// TIA Portal project "chietrotchatlong" (V16)

(* hardware
DEVICE "S7-1200 station_1"  S7-1200 Station
   slot 0: "Rack_0"  S7-1200 Rack  Rack  V1.0
   slot 1: "PLC_1"  CPU 1214C DC/DC/DC  6ES7 214-1AG40-0XB0  V4.4
DEVICE "PC-System_1"  SIMATIC PC station
   slot 0: "SIMATIC PC station"  Rail  SIMATIC PC-Station  V1.0
      slot 125: "Stationmanager"  Station_Manager  V6.0.4
   slot 1: "HMI_RT_1"  WinCC RT Advanced  6AV2 104-0xxxx-xxxx  16.0.0.0
      slot 33792: "Computer interface"  Host interface
   slot 2: "IE general_1"  IE General  IE_CP  V8.2.0
*)

// ===== PLC "PLC_1"  CPU 1214C DC/DC/DC =====

VAR_GLOBAL   // PLC tag table "Default tag table"
   "a0" AT %M0.0 : Bool;
   "a1" AT %M0.1 : Bool;
   "b0" AT %M0.2 : Bool;
   "b1" AT %M0.3 : Bool;
   "d1" AT %M0.4 : Bool;
   "d2" AT %M0.5 : Bool;
   "d3" AT %M0.6 : Bool;
   "g" AT %M0.7 : Bool;
   "S0" AT %Q0.0 : Bool;
   "S1" AT %Q0.1 : Bool;
   "S2" AT %Q0.2 : Bool;
   "S3" AT %Q0.3 : Bool;
   "S4" AT %Q0.4 : Bool;
   "S5" AT %Q0.5 : Bool;
   "S6" AT %Q0.6 : Bool;
   "S7" AT %Q0.7 : Bool;
   "S8" AT %Q1.0 : Bool;
   "m" AT %M1.0 : Bool;
   "ThoiGian" AT %MD1 : Time;
   "START" AT %M1.1 : Bool;
   "STOP" AT %M1.2 : Bool;
   "POWER" AT %Q1.1 : Bool;
END_VAR

// folder: System blocks/Program resources

DATA_BLOCK "T2"   // DB2
{ S7_Optimized_Access := 'TRUE' }
AUTHOR : Simatic
FAMILY : IEC
NAME : IEC_TMR
VERSION : 1.0
// stored: InstanceOfName IEC_TIMER
"IEC_TIMER"
BEGIN
END_DATA_BLOCK

// folder: (top level)

ORGANIZATION_BLOCK "Main"   // OB1, FBD, ProgramCycle
TITLE = "Main Program Sweep (Cycle)"
{ S7_Optimized_Access := 'TRUE' }
VERSION : 0.1
   VAR_INPUT
      Initial_Call : Bool;   // Initial call of this OB
      Remanence : Bool;   // =True, if remanent data are available
   END_VAR
BEGIN

REGION Network 1
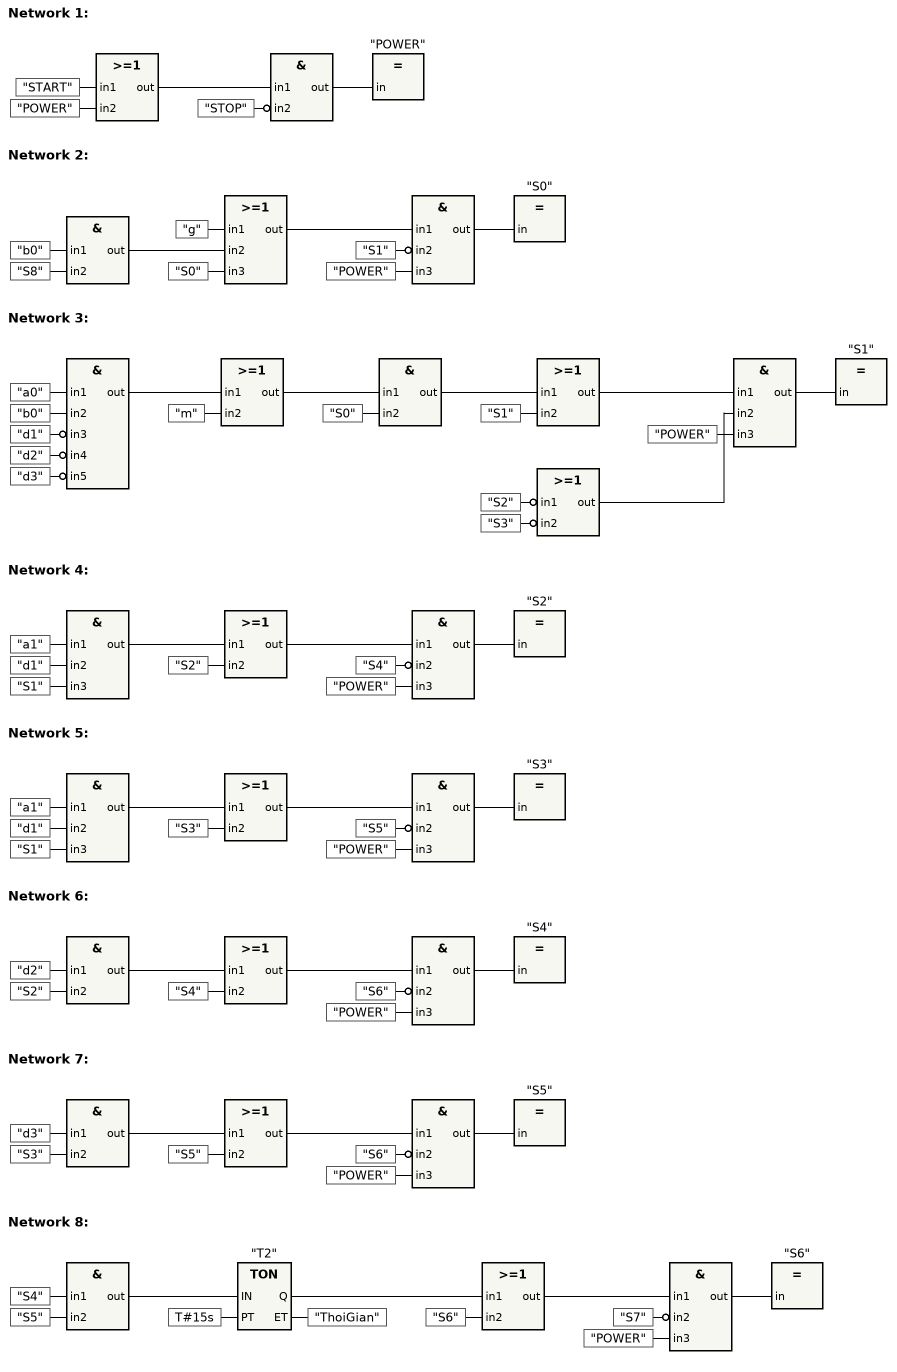
   "POWER" := ("START" OR "POWER") AND NOT "STOP";
END_REGION

REGION Network 2
   "S0" := ("g" OR ("b0" AND "S8") OR "S0") AND NOT "S1" AND "POWER";
END_REGION

REGION Network 3
   "S1" := (((("a0" AND "b0" AND NOT "d1" AND NOT "d2" AND NOT "d3") OR "m") AND "S0") OR "S1") AND (NOT "S2" OR NOT "S3") AND "POWER";
END_REGION

REGION Network 4
   "S2" := (("a1" AND "d1" AND "S1") OR "S2") AND NOT "S4" AND "POWER";
END_REGION

REGION Network 5
   "S3" := (("a1" AND "d1" AND "S1") OR "S3") AND NOT "S5" AND "POWER";
END_REGION

REGION Network 6
   "S4" := (("d2" AND "S2") OR "S4") AND NOT "S6" AND "POWER";
END_REGION

REGION Network 7
   "S5" := (("d3" AND "S3") OR "S5") AND NOT "S6" AND "POWER";
END_REGION

REGION Network 8
   "T2".TON(IN := "S4" AND "S5", PT := T#15s, ET => "ThoiGian");
   "S6" := ("T2".Q OR "S6") AND NOT "S7" AND "POWER";
END_REGION

REGION Network 9
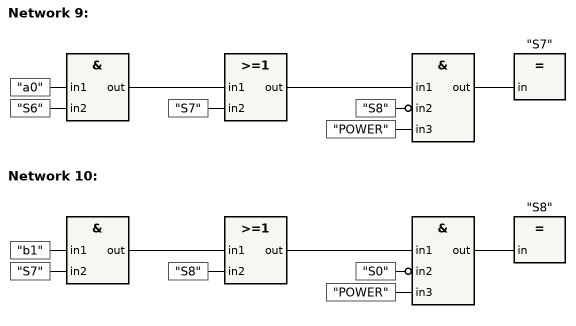
   "S7" := (("a0" AND "S6") OR "S7") AND NOT "S8" AND "POWER";
END_REGION

REGION Network 10
   "S8" := (("b1" AND "S7") OR "S8") AND NOT "S0" AND "POWER";
END_REGION
END_ORGANIZATION_BLOCK

(* ===== HMI "HMI_RT_1" =====
system functions are stored by id; their names below are inferred from use
connection "HMI_Connection_1": ETHERNET, S7_1200_OMS

HMI tags "Default tag table"
   "POWER" : Bool = PLC POWER AT %Q1.1, 1 s
   "S0" : Bool = PLC S0 AT %Q0.0, 1 s
   "S1" : Bool = PLC S1 AT %Q0.1, 1 s
   "S2" : Bool = PLC S2 AT %Q0.2, 1 s
   "S3" : Bool = PLC S3 AT %Q0.3, 1 s
   "S4" : Bool = PLC S4 AT %Q0.4, 1 s
   "S5" : Bool = PLC S5 AT %Q0.5, 1 s
   "S6" : Bool = PLC S6 AT %Q0.6, 1 s
   "S7" : Bool = PLC S7 AT %Q0.7, 1 s
   "S8" : Bool = PLC S8 AT %Q1.0, 1 s
   "START" : Bool = PLC START AT %M1.1, 1 s
   "STOP" : Bool = PLC STOP AT %M1.2, 1 s
   "a0" : Bool = PLC a0 AT %M0.0, 1 s
   "a1" : Bool = PLC a1 AT %M0.1, 1 s
   "b0" : Bool = PLC b0 AT %M0.2, 1 s
   "b1" : Bool = PLC b1 AT %M0.3, 1 s
   "d1" : Bool = PLC d1 AT %M0.4, 1 s
   "d2" : Bool = PLC d2 AT %M0.5, 1 s
   "d3" : Bool = PLC d3 AT %M0.6, 1 s
   "g" : Bool = PLC g AT %M0.7, 1 s
   "m" : Bool = PLC m AT %M1.0, 1 s
   "ThoiGian" : Time = PLC ThoiGian AT %MD1, 1 s

screen "Screen_1" 1024x768
   GraphicView "Graphic view_1" at 255,236 size 64x85; Picture "Graphic_20"
      Visibility <- "S0"
   GraphicView "Graphic view_7" at 383,148 size 56x129; Picture "Graphic_17"
      Visibility <- "S7"
   GraphicView "Graphic view_5" at 149,253 size 166x49; Picture "Graphic_14"
      Visibility <- "S1"
   Rectangle "Rectangle_1" at 721,6 size 57x26
      Appearance <- "POWER"
   Button "Button_1" at 28,15 size 64x33; TextOff 'START'
      on Press: SetBit("START")
      on Release: ResetBit("START")
   Button "Button_2" at 28,61 size 64x33; TextOff 'STOP'
      on Press: SetBit("STOP")
      on Release: ResetBit("STOP")
   Button "Button_3" at 28,107 size 64x33; TextOff 'a0'
      on Press: SetBit("a0")
      on Release: ResetBit("a0")
   Button "Button_4" at 28,153 size 64x33; TextOff 'a1'
      on Release: ResetBit("a1")
      on Press: SetBit("a1")
   Button "Button_5" at 28,199 size 64x33; TextOff 'b0'
      on Activate: SetBit("b0")
      on Deactivate: ResetBit("b0")
   Button "Button_6" at 28,245 size 64x33; TextOff 'b1'
      on Release: ResetBit("b1")
      on Press: SetBit("b1")
   Button "Button_7" at 28,291 size 64x33; TextOff 'd1'
      on Activate: SetBit("d1")
      on Deactivate: ResetBit("d1")
   Button "Button_8" at 28,337 size 64x33; TextOff 'd2'
      on Activate: SetBit("d2")
      on Deactivate: ResetBit("d2")
   Button "Button_9" at 28,383 size 64x33; TextOff 'd3'
      on Activate: SetBit("d3")
      on Deactivate: ResetBit("d3")
   Rectangle "Rectangle_2" at 721,48 size 57x26
      Appearance <- "S0"
   Rectangle "Rectangle_3" at 721,90 size 57x26
      Appearance <- "S1"
   Rectangle "Rectangle_4" at 721,132 size 57x26
      Appearance <- "S2"
   Rectangle "Rectangle_5" at 721,174 size 57x26
      Appearance <- "S3"
   Rectangle "Rectangle_6" at 721,216 size 57x26
      Appearance <- "S4"
   Rectangle "Rectangle_7" at 721,258 size 57x26
      Appearance <- "S5"
   Rectangle "Rectangle_8" at 721,300 size 57x26
      Appearance <- "S6"
   Rectangle "Rectangle_9" at 721,342 size 57x26
      Appearance <- "S7"
   Rectangle "Rectangle_10" at 721,384 size 57x26
      Appearance <- "S8"
   TextField "Text field_1" at 716,6 size 62x22; Text 'POWER'
   TextField "Text field_2" at 737,48 size 25x22; Text 'S0'
   TextField "Text field_3" at 737,91 size 25x22; Text 'S1'
   TextField "Text field_4" at 737,132 size 25x22; Text 'S2'
   TextField "Text field_5" at 737,177 size 25x22; Text 'S3'
   TextField "Text field_6" at 736,218 size 25x22; Text 'S4'
   TextField "Text field_7" at 736,262 size 25x22; Text 'S5'
   TextField "Text field_8" at 736,302 size 25x22; Text 'S6'
   TextField "Text field_9" at 736,346 size 25x22; Text 'S7'
   TextField "Text field_10" at 736,388 size 25x22; Text 'S8'
   Button "Button_10" at 28,430 size 64x33; TextOff 'g'
      on Release: ResetBit("g")
      on Press: SetBit("g")
   Button "Button_11" at 28,477 size 64x33; TextOff 'm'
      on Release: ResetBit("m")
      on Press: SetBit("m")
   GraphicView "Graphic view_4" at 127,250 size 125x50; Picture "Graphic_13"
      Visibility <- "POWER"
   GraphicView "Graphic view_16" at 386,103 size 53x120; Picture "Graphic_15"
      Visibility <- "POWER"
   Circle "Circle_1" at 611,192 size 40x40
      Appearance <- "d3"
   Circle "Circle_2" at 611,236 size 40x40
      Appearance <- "d2"
   Circle "Circle_3" at 611,278 size 40x40
      Appearance <- "d1"
   TextField "Text field_11" at 153,223 size 70x22; Text 'Xi lanh A'
   TextField "Text field_12" at 378,70 size 70x22; Text 'Xi lanh B'
   TextField "Text field_13" at 560,131 size 133x22; Text 'Các đèn cảm biến'
   GraphicView "Graphic view_2" at 376,233 size 64x85; Picture "Graphic_20"
      Visibility <- "S1"
   GraphicView "Graphic view_3" at 376,233 size 64x85; Picture "Graphic_20"
      Visibility <- "S2"
   GraphicView "Graphic view_8" at 376,233 size 64x85; Picture "Graphic_20"
      Visibility <- "S4"
   GraphicView "Graphic view_9" at 376,233 size 64x85; Picture "Graphic_20"
      Visibility <- "S5"
   TextField "Text field_14" at 452,142 size 47x22; Text 'Van C'
   TextField "Text field_15" at 315,152 size 46x22; Text 'Van E'
   GraphicView "Graphic view_12" at 287,177 size 90x59; Picture "Graphic_21"
      Appearance <- "S3"
   GraphicView "Graphic view_13" at 442,171 size 75x66; Picture "Graphic_22"
      Appearance <- "S2"
   GraphicView "Graphic view_14" at 230,202 size 60x31; Picture "Graphic_30"
   GraphicView "Graphic view_15" at 230,1 size 58x204; Picture "Graphic_31"
   GraphicView "Graphic view_17" at 512,177 size 56x75; Picture "Graphic_32"
   GraphicView "Graphic view_18" at 511,0 size 59x181; Picture "Graphic_31"
   GraphicView "Graphic view_19" at 375,346 size 64x85; Picture "Graphic_33"
      Visibility <- "S7"
   GraphicView "Graphic view_11" at 375,346 size 64x85; Picture "Graphic_33"
      Visibility <- "S8"
   GraphicView "Graphic view_20" at 376,233 size 64x85; Picture "Graphic_7"
      Visibility <- "S3"
   GraphicView "Graphic view_21" at 376,233 size 64x85; Picture "Graphic_8"
      Visibility <- "S4"
   GraphicView "Graphic view_22" at 376,233 size 64x85; Picture "Graphic_9"
      Visibility <- "S5"
   GraphicView "Graphic view_6" at 376,233 size 64x85; Picture "Graphic_33"
      Visibility <- "S6"
   TextField "Text field_16" at 568,200 size 24x22; Text 'd3'
   TextField "Text field_17" at 569,239 size 24x22; Text 'd2'
   TextField "Text field_18" at 570,278 size 24x22; Text 'd1'
   TextField "Text field_19" at 569,348 size 113x22; Text 'Thời gian khóa'
   IOField "I/O field_1" at 582,378 size 96x32; FormatPattern 9999999999
      ProcessValue <- "ThoiGian"
*)